FUNCTION_BLOCK Test_WriteBySymbolName_KeepingHandle EXTENDS TUnitTestBase
VAR
    AdsWriteBySymbolName : TAdsWriteBySymbolName;
    ValueToWrite : INT := 3456;
    WriteResult : INT;
    ScanCount : DINT;
    State: INT;
END_VAR

CASE State OF
    0:
        ValueToWrite := 3456;
        WriteResult := 0;
        ScanCount := 0;
    
        AdsWriteBySymbolName.Execute(
            AmsNetId:= '', 
            Port:= 851, 
            SymbolName:= 'PB_TestRunner.Test_WriteBySymbolName_KeepingHandle.WriteResult', 
            WriteDataAddress:= ADR(ValueToWrite), 
            WriteDataLength:= SIZEOF(ValueToWrite), 
            KeepSymbolHandle:= TRUE);
        Test_Started();
        State := 10;
        
    10:
        ScanCount := ScanCount + 1;
        IF NOT AdsWriteBySymbolName.ExecutionResult.Busy THEN
            State := 20;    
		END_IF
        
    20:
        Assertion.AssertEquals_INT(
            Expected     := 3456,
            Actual       := WriteResult,
            ObjectName   := _TestName,
            Variablename := 'WriteResult'); 
 
        Test_Finished();
        State := 0;
END_CASE

AdsWriteBySymbolName();

END_FUNCTION_BLOCK

(* stored: Version 1.1.0.1, ProductVersion 3.1.4024.3
   POU Test_WriteBySymbolName_KeepingHandle: Id {6428be7e-b511-0587-11db-4115f97c9bd2}, SpecialFunc None *)
